FUNCTION_BLOCK FB_Auto_SC
VAR_INPUT
	bEnable				: BOOL;
END_VAR
VAR_OUTPUT
	fPCV				: LREAL;
	fSCV				: LREAL;
	
END_VAR
VAR
	
//Function Blocks
fbPID_OL_startpos				: FB_PID_Controller;
fbPID_OL_sine				: FB_PID_Controller;

fbDeadband_startpos			: FB_Deadband_Auto;
fbDeadband_sine				: FB_Deadband_Auto_sine;

fbDisplacementControl_IL_startpos	: FB_DisplacementControl_SC;
fbDisplacementControl_IL_sine	: FB_DisplacementControl_SC;

fbDerivator					: FB_Derivator;

fbClock						: FB_Clock;
fbSineActivation			: FB_SineActivation_SC;
fbMUX_selector				: FB_MUX_selector;

fbGain_Chooser_P			: FB_GainChooser;
fbGain_Chooser_I			: FB_GainChooser;
fb_ControlReset_startpos	: FB_ControlReset_SC;
fb_ControlReset_sine		:FB_ControlReset_SC;

//Deadband
fDeadbandComp_out			: LREAL;
fDeadbandComp_out_startpos			: LREAL;

//Outer Loop output
fSC_ClosedLoopSingal		: LREAL;
fOuterLoopError				: LREAL;

//Sine Ref signal
fSineRefSignal_SC			: LREAL;
fWinchVelRefSine			: LREAL;

//Valvesignals
fPCV_set					: LREAL := 1.0;
fPCV_On						: LREAL;
fPCV_Off					: LREAL;

fSCV_startpos				: LREAL;
fSCV_sine					: LREAL;
fSCV_Off					: LREAL;


END_VAR
VAR // added by the converter: edge detectors and wires of the graphical bodies
    _w1 : LREAL;
    _w2 : BOOL;
END_VAR

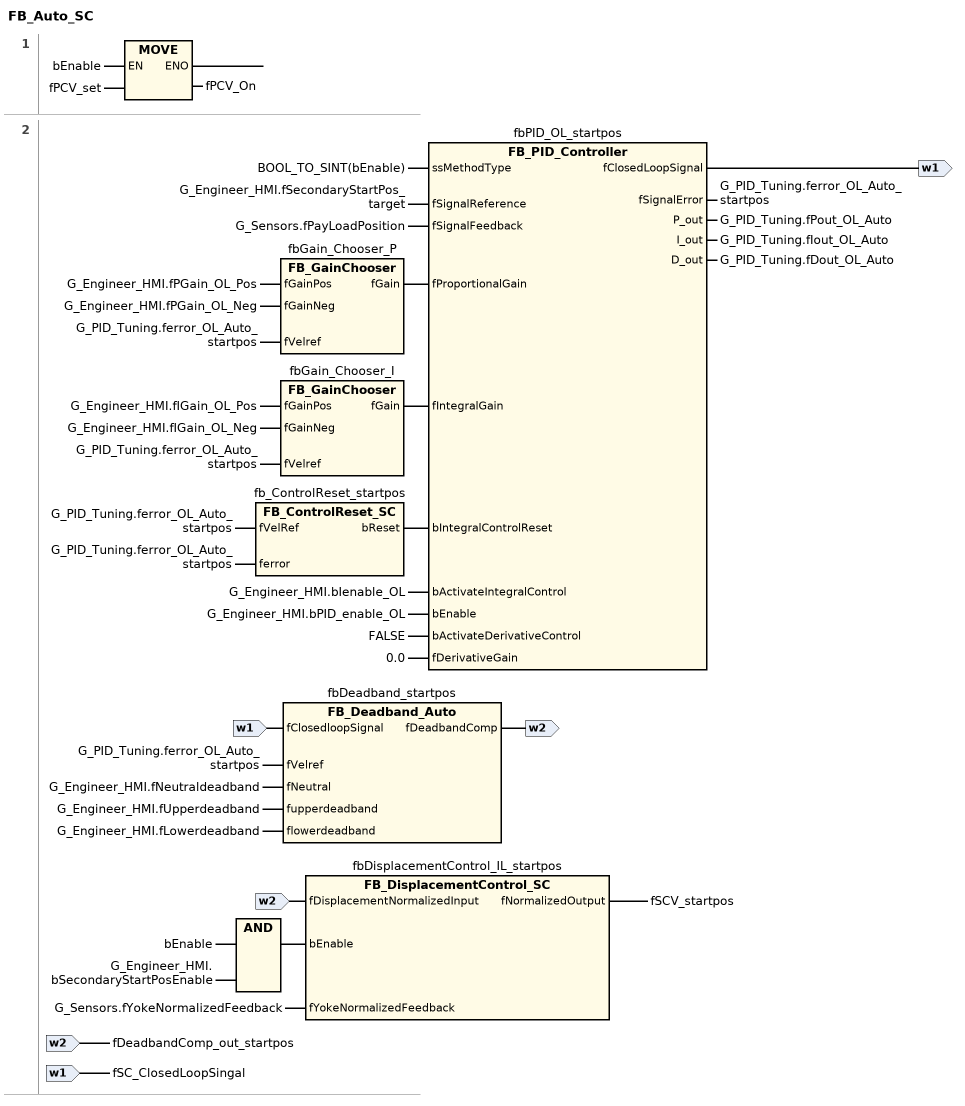
// NETWORK 1
IF bEnable THEN fPCV_On := fPCV_set; END_IF

// NETWORK 2
fbGain_Chooser_P(
    fGainPos := G_Engineer_HMI.fPGain_OL_Pos,
    fGainNeg := G_Engineer_HMI.fPGain_OL_Neg,
    fVelref := G_PID_Tuning.ferror_OL_Auto_startpos); // FB_GainChooser
fbGain_Chooser_I(
    fGainPos := G_Engineer_HMI.fIGain_OL_Pos,
    fGainNeg := G_Engineer_HMI.fIGain_OL_Neg,
    fVelref := G_PID_Tuning.ferror_OL_Auto_startpos); // FB_GainChooser
fb_ControlReset_startpos(fVelRef := G_PID_Tuning.ferror_OL_Auto_startpos, ferror := G_PID_Tuning.ferror_OL_Auto_startpos); // FB_ControlReset_SC
fbPID_OL_startpos(
    ssMethodType := BOOL_TO_SINT(bEnable),
    fSignalReference := G_Engineer_HMI.fSecondaryStartPos_target,
    fSignalFeedback := G_Sensors.fPayLoadPosition,
    fProportionalGain := fbGain_Chooser_P.fGain,
    fIntegralGain := fbGain_Chooser_I.fGain,
    bIntegralControlReset := fb_ControlReset_startpos.bReset,
    bActivateIntegralControl := G_Engineer_HMI.bIenable_OL,
    bEnable := G_Engineer_HMI.bPID_enable_OL,
    bActivateDerivativeControl := FALSE,
    fDerivativeGain := 0.0,
    fSignalError => G_PID_Tuning.ferror_OL_Auto_startpos,
    P_out => G_PID_Tuning.fPout_OL_Auto,
    I_out => G_PID_Tuning.fIout_OL_Auto,
    D_out => G_PID_Tuning.fDout_OL_Auto); // FB_PID_Controller
fbDeadband_startpos(
    fClosedloopSignal := fbPID_OL_startpos.fClosedLoopSignal,
    fVelref := G_PID_Tuning.ferror_OL_Auto_startpos,
    fNeutral := G_Engineer_HMI.fNeutraldeadband,
    fupperdeadband := G_Engineer_HMI.fUpperdeadband,
    flowerdeadband := G_Engineer_HMI.fLowerdeadband); // FB_Deadband_Auto
fbDisplacementControl_IL_startpos(
    fDisplacementNormalizedInput := fbDeadband_startpos.fDeadbandComp,
    bEnable := bEnable AND G_Engineer_HMI.bSecondaryStartPosEnable,
    fYokeNormalizedFeedback := G_Sensors.fYokeNormalizedFeedback); // FB_DisplacementControl_SC
fSCV_startpos := fbDisplacementControl_IL_startpos.fNormalizedOutput;
fDeadbandComp_out_startpos := fbDeadband_startpos.fDeadbandComp;
fSC_ClosedLoopSingal := fbPID_OL_startpos.fClosedLoopSignal;

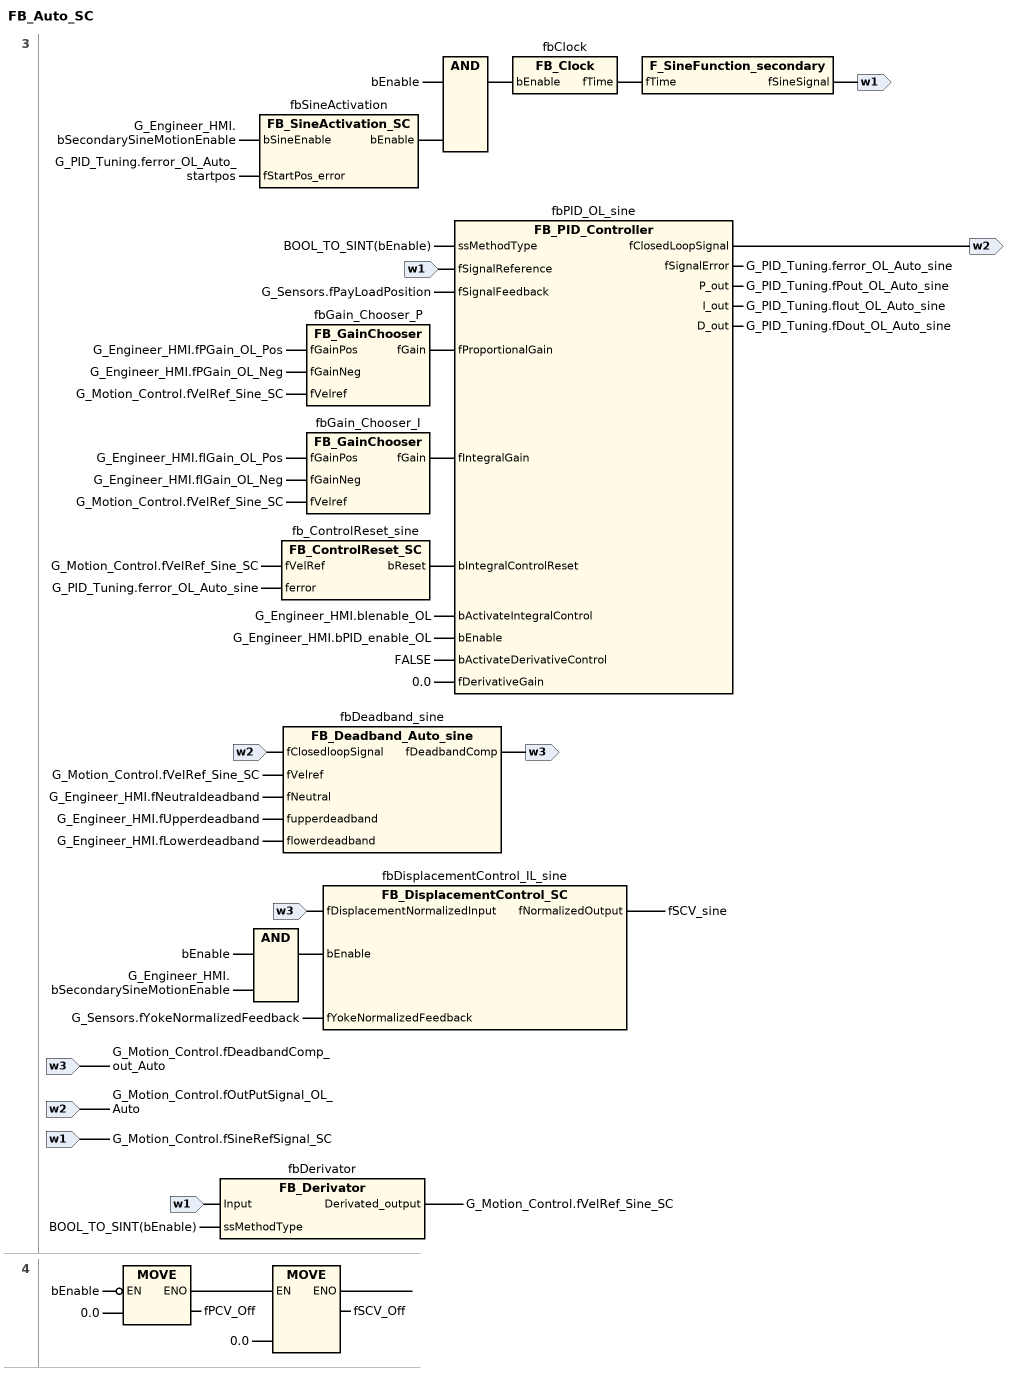
// NETWORK 3
fbSineActivation(bSineEnable := G_Engineer_HMI.bSecondarySineMotionEnable, fStartPos_error := G_PID_Tuning.ferror_OL_Auto_startpos); // FB_SineActivation_SC
fbClock(bEnable := bEnable AND fbSineActivation.bEnable); // FB_Clock
F_SineFunction_secondary(fTime := fbClock.fTime, fSineSignal => _w1);
fbGain_Chooser_P(
    fGainPos := G_Engineer_HMI.fPGain_OL_Pos,
    fGainNeg := G_Engineer_HMI.fPGain_OL_Neg,
    fVelref := G_Motion_Control.fVelRef_Sine_SC); // FB_GainChooser
fbGain_Chooser_I(
    fGainPos := G_Engineer_HMI.fIGain_OL_Pos,
    fGainNeg := G_Engineer_HMI.fIGain_OL_Neg,
    fVelref := G_Motion_Control.fVelRef_Sine_SC); // FB_GainChooser
fb_ControlReset_sine(fVelRef := G_Motion_Control.fVelRef_Sine_SC, ferror := G_PID_Tuning.ferror_OL_Auto_sine); // FB_ControlReset_SC
fbPID_OL_sine(
    ssMethodType := BOOL_TO_SINT(bEnable),
    fSignalReference := _w1,
    fSignalFeedback := G_Sensors.fPayLoadPosition,
    fProportionalGain := fbGain_Chooser_P.fGain,
    fIntegralGain := fbGain_Chooser_I.fGain,
    bIntegralControlReset := fb_ControlReset_sine.bReset,
    bActivateIntegralControl := G_Engineer_HMI.bIenable_OL,
    bEnable := G_Engineer_HMI.bPID_enable_OL,
    bActivateDerivativeControl := FALSE,
    fDerivativeGain := 0.0,
    fSignalError => G_PID_Tuning.ferror_OL_Auto_sine,
    P_out => G_PID_Tuning.fPout_OL_Auto_sine,
    I_out => G_PID_Tuning.fIout_OL_Auto_sine,
    D_out => G_PID_Tuning.fDout_OL_Auto_sine); // FB_PID_Controller
fbDeadband_sine(
    fClosedloopSignal := fbPID_OL_sine.fClosedLoopSignal,
    fVelref := G_Motion_Control.fVelRef_Sine_SC,
    fNeutral := G_Engineer_HMI.fNeutraldeadband,
    fupperdeadband := G_Engineer_HMI.fUpperdeadband,
    flowerdeadband := G_Engineer_HMI.fLowerdeadband); // FB_Deadband_Auto_sine
fbDisplacementControl_IL_sine(
    fDisplacementNormalizedInput := fbDeadband_sine.fDeadbandComp,
    bEnable := bEnable AND G_Engineer_HMI.bSecondarySineMotionEnable,
    fYokeNormalizedFeedback := G_Sensors.fYokeNormalizedFeedback); // FB_DisplacementControl_SC
fSCV_sine := fbDisplacementControl_IL_sine.fNormalizedOutput;
G_Motion_Control.fDeadbandComp_out_Auto := fbDeadband_sine.fDeadbandComp;
G_Motion_Control.fOutPutSignal_OL_Auto := fbPID_OL_sine.fClosedLoopSignal;
G_Motion_Control.fSineRefSignal_SC := _w1;
fbDerivator(Input := _w1, ssMethodType := BOOL_TO_SINT(bEnable)); // FB_Derivator
G_Motion_Control.fVelRef_Sine_SC := fbDerivator.Derivated_output;

// NETWORK 4
_w2 := NOT bEnable;
IF _w2 THEN fPCV_Off := 0.0; END_IF
IF _w2 THEN fSCV_Off := 0.0; END_IF

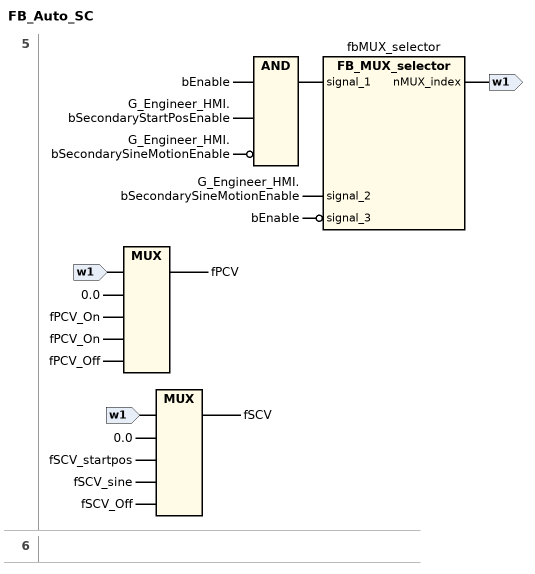
// NETWORK 5
fbMUX_selector(
    signal_1 := bEnable AND G_Engineer_HMI.bSecondaryStartPosEnable AND NOT G_Engineer_HMI.bSecondarySineMotionEnable,
    signal_2 := G_Engineer_HMI.bSecondarySineMotionEnable,
    signal_3 := NOT bEnable); // FB_MUX_selector
fPCV := MUX(fbMUX_selector.nMUX_index, 0.0, fPCV_On, fPCV_On, fPCV_Off);
fSCV := MUX(fbMUX_selector.nMUX_index, 0.0, fSCV_startpos, fSCV_sine, fSCV_Off);

// NETWORK 6

END_FUNCTION_BLOCK

(* stored: Version 1.1.0.1
   POU FB_Auto_SC: Id {376f8971-d678-4d52-b268-171162ccc33c}, SpecialFunc None *)
